# B&R Automation Studio project Tires_Krichev
Automation Studio 3.0.90.25 SP07; Krichev. Equipment tire burning


## Configuration Simulation

### Task classes (Cpu.sw)
```
Cyclic#2:
  spreading <- spreading.prg
  Conv_mitsu <- Conv_mitsubishi.prg [disabled]
  Sleep <- Sleep.prg
  manualCont <- manualControl.prg
  autoContro <- autoControl.prg
  weightCont <- weightControl.prg
  modbusRTU <- modbusRTU.prg
Cyclic#3:
  TechProces <- TechProcess.prg
  visual <- visual.prg
Cyclic#4:
  exampleCpl <- exampleCplusplus.prg [disabled]
DataObjects: Arnc0sys, Acp10sys
NcDataObjects: gmcipsys <- GmcIpConfig.gmcipsys.dob, gmciplbr <- GmcIpConfig.gmciplbr.dob, gmcipcbr <- GmcIpConfig.gmcipcbr.dob, gmciplsm <- GmcIpConfig.gmciplsm.dob, gmcipcsm <- GmcIpConfig.gmcipcsm.dob, gmcipcfg <- GmcIpConfig.gmcipcfg.dob, gmcipiec <- GmcIpConfig.gmcipiec.dob, gmciplog <- GmcIpConfig.gmciplog.dob, gmcipvar <- GmcIpUserConfig.gmcipvar.dob, gmcipfun <- GmcIpUserConfig.gmcipfun.dob, gmcipfub <- GmcIpUserConfig.gmcipfub.dob, gmcipubr <- GmcIpUserConfig.gmcipubr.dob, gmcipusm <- GmcIpUserConfig.gmcipusm.dob
VcDataObjects: Visu <- Visu.dob
Binaries: vccbar, visvc, Visu01, Visu02, vcfntttf, vccshape, vcctext, vccovl, arial, vctcal, vccbtn, vccnum, vcpfar00, vcdsint, vcpdvnc, vcpdsw, vcalarm, vcchspot, vcfile, vcmgr, vccstr, vcresman, vcgclass, vcdsloc, arialbd, vcnet, vcrt, vccalarm, vcclbox, vccbmp, vcbclass, vcshared, vccline, vcctrend, Visu03, Arnc0cfg, Acp10cfg, ashwd, arconfig, sysconf, asfw, iomap
Libraries: AsIecCon, astime, visapi, fileio, dataobj, runtime, standard, dvframe, Arnc0man, AsMem, AsArLog, Acp10man, sys_lib, AsArProf, brsystem, NcGlobal, Acp10par, powerlnk
```

### Acp10cfg.ncc - PLC1/Motion/Acp10cfg.ncc
```
NcConfiguration (Version=2.28.2, NcSwId=acp10)
  ACP10CF1_typ:
    cnt_nettrc_rec_drive = 1500
    bufsize_trace_upload = 1200
    tc_nc_man_task = Cyclic #1
    glob_pv_as_ncobject = Yes
    network_init:
      ncsw_init_execute = Yes
      automatic_execute = No
      node_nr_warning = Yes
      net_err_before_ncact = Yes
    nettrc:
      enter_parsecrec = Yes
      enter_ncaction = Yes
      save_ring_startidx = Yes
```

### Arnc0cfg.ncc - PLC1/Motion/Arnc0cfg.ncc
```
NcConfiguration (Version=1.28.1, NcSwId=arnc0)
  ARNC0CFG_typ:
    sampling_rate = 4000
    cnt_nettrc_rec_drive = 1500
    bufsize_sys_trace = 16#00005000
    enable_mp_log = Yes
    tc_nc_man_task = Cyclic #1
    bg_load = 1
    glob_pv_as_ncobject = Yes
```

## Configuration config

### Task classes (Cpu.sw)
```
Cyclic#4:
  visual <- visual.prg
  TechProces <- TechProcess.prg
  Conv_mitsu <- Conv_mitsubishi.prg [disabled]
  weightCont <- weightControl.prg
  manualCont <- manualControl.prg
  autoContro <- autoControl.prg
  spreading <- spreading.prg
  modbusRTU <- modbusRTU.prg [disabled]
Cyclic#5:
  Sleep <- Sleep.prg
NcDataObjects: gmcipsys <- GmcIpConfig.gmcipsys.dob, gmciplbr <- GmcIpConfig.gmciplbr.dob, gmcipcbr <- GmcIpConfig.gmcipcbr.dob, gmciplsm <- GmcIpConfig.gmciplsm.dob, gmcipcsm <- GmcIpConfig.gmcipcsm.dob, gmcipcfg <- GmcIpConfig.gmcipcfg.dob, gmcipiec <- GmcIpConfig.gmcipiec.dob, gmciplog <- GmcIpConfig.gmciplog.dob, gmcipvar <- GmcIpUserConfig.gmcipvar.dob, gmcipfun <- GmcIpUserConfig.gmcipfun.dob, gmcipfub <- GmcIpUserConfig.gmcipfub.dob, gmcipubr <- GmcIpUserConfig.gmcipubr.dob, gmcipusm <- GmcIpUserConfig.gmcipusm.dob
VcDataObjects: Visu <- Visu.dob
Binaries: vccalarm, vcclbox, vcctext, vcrt, vcchspot, vcpdpp30, vccbar, vcresman, vcpfmtcx, vcptelo, vcfile, vcdsint, vcpdsw, vccshape, arial, vccbmp, vcmgr, Visu01, vcctrend, vcfntttf, vcgclass, vccovl, vctcal, arialbd, vcalarm, vccnum, vccline, vcshared, vcdsloc, vccbtn, vccstr, vcbclass, vcpfpp30, Visu03, Visu02, arconfig, sysconf, ashwd, asfw, iomap
Libraries: fileio, standard, astime, runtime, dataobj, dvframe
```

## Configuration master

### Task classes (Cpu.sw)
```

```

## Configuration slave

### Task classes (Cpu.sw)
same as Physical/master/PLC1/Cpu.sw

- Physical/slave/PLC1/Cpu.per: same as Physical/master/PLC1/Cpu.per
- Physical/slave/PLC1/IoMap.iom: same as Physical/master/PLC1/IoMap.iom
- Physical/slave/PLC1/PvMap.vvm: same as Physical/master/PLC1/PvMap.vvm
## Logical view

### Global.var - Global variables
```iecst
(********************************************************************
 * COPYRIGHT --
 ********************************************************************
 * File: Global.var
 * Author: vzylevich
 * Created: June 24, 2013
 ********************************************************************
 * Global variables of project Tires_Krichev
 ********************************************************************)
VAR
	b : UINT := 0; (*Отладка*)
	a : UINT := 0; (*Отладка*)
	maxTireWeight : USINT := 0; (*Максимальный вес шины*)
	minTireWeight : USINT := 0; (*Минимальный вес шины*)
	pulseSignal : USINT := 0; (*Индикатор запуска пульсирующего сигнала технологического светофора*)
	sensSB4Light : USINT := 0; (*Лампа на кнопке SB4*)
	mod : USINT := 0;
	TON_count : TON := (0);
	TON0 : TON := (0);
	TON_01 : TON := (0);
	count : USINT := 0; (*Счетчик секунд пульсирующего сигнала (30 сек)*)
	var : USINT := 0; (*Переменная для отображения заголовков рольганга*)
	elmotorM : ARRAY[0..12] OF USINT := [13(0)]; (*Массив для электродвигателей*)
	sensRemoteControl : ARRAY[0..13] OF USINT := [14(1)]; (*Массив для датчиков дистанционного управления*)
	sensLocalControl : ARRAY[0..13] OF USINT := [14(0)]; (*Массив для датчиков местного управления (пуск).*)
	sensSQAlarm : ARRAY[0..6] OF USINT := [5(0)]; (*Датчики аварийных предупреждений*)
	sensSQ : ARRAY[0..14] OF USINT := [13(0)]; (*Массив для датчиков положения покрышки на рольгангах и конвейерах.*)
	modeControl : USINT := 0; (*Режим управления*)
	tireWeightRolg7 : USINT := 0; (*Вес шины на рольганге 7*)
	lineCapacityMin : UINT := 0; (*Минимальная производительность линии*)
	lineCapacityMax : UINT := 0; (*Максимальная производительность линии*)
	transporterSpeed : USINT := 0; (*Скорость транспортера*)
	tireWeightMin : USINT := 0; (*Минимальный вес шины, загружаемой на конвейер 8*)
	tireWeightMax : USINT := 0; (*Максимальный вес шины, загружаемой на конвейер 8*)
	furnReady : USINT := 0; (*Готовность печи*)
	tireWeightRolg6 : USINT := 0; (*Вес шины на рольганге 6*)
	tireWeightConv8 : USINT := 0; (*Вес шины на конвейере 8*)
	resValueTires : USINT := 0; (*Остаточное значение шин*)
	realCapacity : USINT := 0; (*Действительное значение производительности*)
	nomCapacity : UINT := 0; (*Номинальное значние производительности*)
	scalesMSG : USINT := 0; (*Сообщение "Весы готовы"*)
	sensSB4 : USINT := 0; (*Датчик автоматического режима управления*)
	sensHL12 : USINT := 0; (*Датчик ручного режима управления*)
	sensY2 : USINT := 0;
	sensY1 : USINT := 0;
END_VAR
(*Датчики*)
VAR
	sensSQ70 : USINT := 0;
	sensSQ68 : USINT := 0;
	sensSQ67 : USINT := 0;
	sensSQ66 : USINT := 0;
	sensSQ65 : USINT := 0;
	sensSQ64 : USINT := 0;
	sensSQ62 : USINT := 0;
	sensSQ51 : USINT := 0;
	sensSQ49 : USINT := 0;
	sensSQ48 : USINT := 0;
	sensSQ46 : USINT := 0;
	sensSQ44 : USINT := 0;
	sensSQ43 : USINT := 0;
	sensSQ42 : USINT := 0;
	sensSQ24 : USINT := 0;
END_VAR
```

- Visualisation Logical/Visu (not shown)

- Visualisation Logical/visual (not shown)

### Program Logical/TechProcess (ANSIC) - the description line work tire burning

#### modesControl.h
```c
/********************************************************************
 * COPYRIGHT --
 ********************************************************************
 * Program: TechProcess
 * File: modesControl.h
 * Author: VZylevich
 * Created: July 05, 2013
 *******************************************************************/

#include <bur/plctypes.h>

#ifdef _DEFAULT_INCLUDES
	#include <AsDefault.h>
#endif

/*Количество датчиков местного управления*/
USINT amountModeControl()
{
	return sizeof(sensRemoteControl);
}

USINT amountSensAlarm()
{
	return sizeof(sensSQAlarm);
}

/*Проверка условий останова автоматического режима*/
BOOL checkAutoStop(USINT array[], USINT numOfElements, BOOL onOff)
{
	for (i = 0; i < numOfElements; i++)
	{
		if (array[i] == onOff)
		{
			checkStop = 0;
			sensSB4 = 0;
			sensSB4Light = 0;
			count = 0;
			TON_count.IN = 0;
			TON_count.ET = 0;
			TON_count.StartTime = 0;
			break;
		}
		else checkStop = 1;
	}
	return checkStop;
}

/*Проверка условий и запуск автоматического режима управления*/
int checkAutoMode()
{
	rControl = checkAutoStop(sensRemoteControl, amountModeControl(), 0);
	sensAlarm = checkAutoStop(sensSQAlarm, amountSensAlarm(), 1);

	if (sensSB4 && rControl && sensAlarm)
	{
		(TON_count.ET < 30000) ? (pulseSignal = 1) : (pulseSignal = 0);	//Пульсирующий сигнал техн. светофоров
		autoMode = 1;
	}
	else
	{
		sensSB4Light = 0;
		count = 0;
		TON_count.IN = 0;
		TON_count.ET = 0;
		TON_count.StartTime = 0;
		autoMode = 0;
	}
	return autoMode;
}

/*Проверка условий и запуск ручного режима управления*/
int checkManMode()
{
	ssModeControl = amountModeControl();
	if (sensHL12 == 1)
	{
		for (i = 0; i < ssModeControl; i++)
			sensLocalControl[i] = 1;
		manMode = 1;
		if (checkAutoMode())
		{
			for (i = 0; i < ssModeControl; i++)
				sensRemoteControl[i] = 0;
			sensSB4 = 0;
			rControl = 0;
			autoMode = 0;
		}
	} else{
		for (i = 0; i < ssModeControl; i++)
			sensLocalControl[i] = 0;
		manMode = 0;
	}
	return manMode;
}

/*int autoMode()
{
	sensSQ[0] ?
	return 0;
}*/
```

#### TechProcess.c - Cyclic code
```c
/********************************************************************
 * COPYRIGHT --
 ********************************************************************
 * Program: TechProcess
 * File: TechProcess.c
 * Author: VZylevich
 * Created: July 02, 2013
 ********************************************************************
 * Implementation of program TechProcess
 ********************************************************************/
#include <bur/plctypes.h>
#include <standard.h>
#include "modesControl.h"

#ifdef _DEFAULT_INCLUDES
	#include <AsDefault.h>
#endif

void _CYCLIC TechProcess(void)
{
	if (checkManMode())
	{
		timeStruct.second = 0;
		foo = 0;
	}
	else if (checkAutoMode())
	{

	}
}
```

#### TechProcess.var - Local variables
```iecst
(********************************************************************
 * COPYRIGHT --
 ********************************************************************
 * Program: TechProcess
 * File: TechProcess.var
 * Author: VZylevich
 * Created: July 02, 2013
 ********************************************************************
 * Local variables of program TechProcess
 ********************************************************************)
VAR
	checkStop : BOOL := FALSE;
	sensAlarm : USINT := 0; (*Датчик предупреждения*)
	rControl : USINT := 0;
	ssModeControl : USINT := 0;
	autoMode : BOOL := FALSE;
	manMode : BOOL := FALSE;
	timeStruct : TIMEStructure := (0);
	foo : UINT := 0; (*Отладка*)
	i : USINT := 0;
END_VAR
```

### Program Logical/Sleep (ANSIC) - A new program

#### Sleep.c - Cyclic code
```c
/********************************************************************
 * COPYRIGHT --
 ********************************************************************
 * Program: Sleep
 * File: Sleep.c
 * Author: VZylevich
 * Created: July 10, 2013
 ********************************************************************
 * Implementation of program Sleep
 ********************************************************************/

#include <bur/plctypes.h>

#ifdef _DEFAULT_INCLUDES
	#include <AsDefault.h>
#endif

_LOCAL USINT i;
_LOCAL USINT foo;

/*Пульсирующий сигнал технологических светофоров длительностью 30 секунд*/
void timerAutoMode(void)
{
	if (sensSB4)
	{
		if(pulseSignal)
		{
			TON_count.IN = !TON_count.Q;
			TON_count.PT = 30000;
			TON(&TON_count);
			if(TON_count.ET < 30000)
			{
				pulseSignal = 1;
				TON_01.IN = !TON_01.Q;
				TON_01.PT = 1000;
				TON(&TON_01);
				count = TON_count.ET / TON_01.PT;
				(count % 2) ? (sensSB4Light = 0) : (sensSB4Light = 1);
			} else
			{
				sensSB4Light = 1;
				pulseSignal = 0;
			}
		}
	}
}

/*Моделирование передвижения шин по конвейеру*/
void tireMoving()
{
	if(foo)
	{
		if(i < sizeof(sensSQ))
		{
			if(i > 0) sensSQ[i-1] = 0;
			sensSQ[i] = 1;
			(i % 2) ? (TON0.IN = 1) : (TON0.IN = 0);
			TON0.PT = 5000;
			TON(&TON0);
			i++;
		}else i = 0;
	}else for(i = 0; i < sizeof(sensSQ); i++)
			sensSQ[i] = 0;
}

void _CYCLIC Sleep(void)
{
	timerAutoMode();
	tireMoving();
}
```

### Program Logical/manualControl (ANSIC) - A new program

#### manualControl.c - Cyclic code
```c
/********************************************************************
 * COPYRIGHT --
 ********************************************************************
 * Program: manualControl
 * File: manualControl.c
 * Author: VZylevich
 * Created: July 15, 2013
 ********************************************************************
 * Implementation of program manualControl
 ********************************************************************/

#include <bur/plctypes.h>

#ifdef _DEFAULT_INCLUDES
	#include <AsDefault.h>
#endif

void _CYCLIC manualControl(void)
{
	/* TODO: Add code here */
}
```

#### modesControl.h
```c
/********************************************************************
 * COPYRIGHT --
 ********************************************************************
 * Program: TechProcess
 * File: modesControl.h
 * Author: VZylevich
 * Created: July 05, 2013
 *******************************************************************/

#include <bur/plctypes.h>

#ifdef _DEFAULT_INCLUDES
	#include <AsDefault.h>
#endif

/*Количество датчиков местного управления*/
USINT amountModeControl()
{
	return sizeof(sensRemoteControl);
}

USINT amountSensAlarm()
{
	return sizeof(sensSQAlarm);
}

/*Проверка условий останова автоматического режима*/
BOOL checkAutoStop(USINT array[], USINT numOfElements, BOOL onOff)
{
	for (i = 0; i < numOfElements; i++)
	{
		if (array[i] == onOff)
		{
			checkStop = 0;
			sensSB4 = 0;
			sensSB4Light = 0;
			count = 0;
			TON_count.IN = 0;
			TON_count.ET = 0;
			TON_count.StartTime = 0;
			break;
		}
		else checkStop = 1;
	}
	return checkStop;
}

/**/
int checkManMode()
{
	ssModeControl = amountModeControl();
	if (sensHL12 == 1)
	{
		for (i = 0; i < ssModeControl; i++)
			sensLocalControl[i] = 1;
		manMode = 1;
		if (checkAutoMode())
		{
			for (i = 0; i < ssModeControl; i++)
				sensRemoteControl[i] = 0;
			sensSB4 = 0;
			rControl = 0;
			autoMode = 0;
		}
	} else{
		for (i = 0; i < ssModeControl; i++)
			sensLocalControl[i] = 0;
		manMode = 0;
	}
	return manMode;
}

/**/
int checkAutoMode()
{
	rControl = checkAutoStop(sensRemoteControl, amountModeControl(), 0);
	sensAlarm = checkAutoStop(sensSQAlarm, amountSensAlarm(), 1);

	if (sensSB4 && rControl && sensAlarm)
	{
		(TON_count.ET < 30000) ? (pulseSignal = 1) : (pulseSignal = 0);
		autoMode = 1;
	}
	else
	{
		sensSB4Light = 0;
		count = 0;
		TON_count.IN = 0;
		TON_count.ET = 0;
		TON_count.StartTime = 0;
		autoMode = 0;
	}
	return autoMode;
}

/*int autoMode()
{
	sensSQ[0] ?
	return 0;
}*/
```

### Program Logical/autoControl (ANSIC) - A new program

#### autoControl.c - Cyclic code
```c
/********************************************************************
 * COPYRIGHT --
 ********************************************************************
 * Program: autoControl
 * File: autoControl.c
 * Author: VZylevich
 * Created: July 15, 2013
 ********************************************************************
 * Implementation of program autoControl
 ********************************************************************/

#include <bur/plctypes.h>

#ifdef _DEFAULT_INCLUDES
	#include <AsDefault.h>
#endif

void _CYCLIC autoControl(void)
{
	/* TODO: Add code here */
}
```

#### modesControl.h
```c
/********************************************************************
 * COPYRIGHT --
 ********************************************************************
 * Program: TechProcess
 * File: modesControl.h
 * Author: VZylevich
 * Created: July 05, 2013
 *******************************************************************/

#include <bur/plctypes.h>

#ifdef _DEFAULT_INCLUDES
	#include <AsDefault.h>
#endif

/*Количество датчиков местного управления*/
USINT amountModeControl()
{
	return sizeof(sensRemoteControl);
}

USINT amountSensAlarm()
{
	return sizeof(sensSQAlarm);
}

/*Проверка условий останова автоматического режима*/
BOOL checkAutoStop(USINT array[], USINT numOfElements, BOOL onOff)
{
	for (i = 0; i < numOfElements; i++)
	{
		if (array[i] == onOff)
		{
			checkStop = 0;
			sensSB4 = 0;
			sensSB4Light = 0;
			count = 0;
			TON_count.IN = 0;
			TON_count.ET = 0;
			TON_count.StartTime = 0;
			break;
		}
		else checkStop = 1;
	}
	return checkStop;
}

/**/
int checkManMode()
{
	ssModeControl = amountModeControl();
	if (sensHL12 == 1)
	{
		for (i = 0; i < ssModeControl; i++)
			sensLocalControl[i] = 1;
		manMode = 1;
		if (checkAutoMode())
		{
			for (i = 0; i < ssModeControl; i++)
				sensRemoteControl[i] = 0;
			sensSB4 = 0;
			rControl = 0;
			autoMode = 0;
		}
	} else{
		for (i = 0; i < ssModeControl; i++)
			sensLocalControl[i] = 0;
		manMode = 0;
	}
	return manMode;
}

/**/
int checkAutoMode()
{
	rControl = checkAutoStop(sensRemoteControl, amountModeControl(), 0);
	sensAlarm = checkAutoStop(sensSQAlarm, amountSensAlarm(), 1);

	if (sensSB4 && rControl && sensAlarm)
	{
		(TON_count.ET < 30000) ? (pulseSignal = 1) : (pulseSignal = 0);
		autoMode = 1;
	}
	else
	{
		sensSB4Light = 0;
		count = 0;
		TON_count.IN = 0;
		TON_count.ET = 0;
		TON_count.StartTime = 0;
		autoMode = 0;
	}
	return autoMode;
}

/*int autoMode()
{
	sensSQ[0] ?
	return 0;
}*/
```

### Program Logical/weightControl (ANSIC) - A new program

#### weightControl.c - Cyclic code
```c
/********************************************************************
 * COPYRIGHT --
 ********************************************************************
 * Program: weightControl
 * File: weightControl.c
 * Author: VZylevich
 * Created: July 15, 2013
 ********************************************************************
 * Implementation of program weightControl
 ********************************************************************/

#include <bur/plctypes.h>

#ifdef _DEFAULT_INCLUDES
	#include <AsDefault.h>
#endif
void _INIT inity(void)
{
	a = 0;
	b = 0;
}

TIME rotationPeriod(void)
{
	/*Определяем время оборота печи*/
	if (sensSQ70){
		rotation = 1;
		time ? (period = time) : (period = 0);
	}
	if (!sensSQ70 && rotation)
		time = clock_ms();

	return period;
}

/*Загрузка печи*/
UDINT furnaceLoading(TIME rotationFurnace)
{
	Qrot = (nomCapacity * (UDINT) rotationFurnace) / hour;
	return Qrot;
}

/*Производительность сжигания*/
UDINT capacityBurning(void)
{
	return (nomCapacity * 1000)/ hour;
}

/*Задержка для успокоения весов*/
void delay(USINT sensor)
{
	if (sensor){
		TON_atten.IN = !TON_atten.Q;
		TON_atten.PT = attenuation;
		TON(&TON_atten);
	}
}
void _CYCLIC weightControl(void)
{
	tRot = rotationPeriod();	//Время одного оборота печи
	if (tRot)
		kgRotation = furnaceLoading(tRot); //Определяем кол-во килограмм шин необходимых для загрузки печи за один оборот
	kgSec = capacityBurning();	//Производительносто подачи шин на сжигание в секунду
	delay(sensSQ70);
	(TON_atten.ET == attenuation) ? (weightMeasure = weight) : (weightMeasure = 0);//Если время успокоения прошло, присвоить значение веса
	if (weightMeasure && !sensSQ[7])	//Если известен вес и на рольганге 7 пусто - включить электродвигатель рольганга
		elmotorM[6] = 1;
	if (weightMeasure && sensSQ[7])		//Если известен вес и на рольганге 7 есть шина, передать измерен. знач. веса шины в загрузку
		loadingRollg7 = weightMeasure;

}
```

#### weightControl.var - Local variables
```iecst
(********************************************************************
 * COPYRIGHT --
 ********************************************************************
 * Program: weightControl
 * File: weightControl.var
 * Author: VZylevich
 * Created: July 15, 2013
 ********************************************************************
 * Local variables of program weightControl
 ********************************************************************)
VAR
	kgSec : USINT := 0; (*Производительность печи*)
	period : USINT := 0;
	rotation : USINT := 0;
	loadingRollg7 : USINT := 0; (*Вес шины на позиции загрузки(рольганг 7)*)
	weight : USINT := 0;
	weightMeasure : USINT := 0;
	TON_atten : TON := (0); (*Время необходимое для успокоения весов перед взвешинванием*)
	attenuation : USINT := 0; (*Затухание весов*)
	Qrot : UDINT := 0;
	kgRotation : REAL := 0.0; (*Кол-во кг сжигаемых шин за 1 оборот*)
END_VAR
VAR CONSTANT
	hour : UDINT := 3600000; (*1 час в мс*)
END_VAR
VAR
	time : TIME := T#0S;
	tRot : TIME := T#0S; (*Время оборота печи*)
	(*TON_weightLoading : TON := (0);*)
END_VAR
```

#### modesControl.h
```c
/********************************************************************
 * COPYRIGHT --
 ********************************************************************
 * Program: TechProcess
 * File: modesControl.h
 * Author: VZylevich
 * Created: July 05, 2013
 *******************************************************************/

#include <bur/plctypes.h>

#ifdef _DEFAULT_INCLUDES
	#include <AsDefault.h>
#endif

/*Количество датчиков местного управления*/
USINT amountModeControl()
{
	return sizeof(sensRemoteControl);
}

USINT amountSensAlarm()
{
	return sizeof(sensSQAlarm);
}

/*Проверка условий останова автоматического режима*/
BOOL checkAutoStop(USINT array[], USINT numOfElements, BOOL onOff)
{
	for (i = 0; i < numOfElements; i++)
	{
		if (array[i] == onOff)
		{
			checkStop = 0;
			sensSB4 = 0;
			sensSB4Light = 0;
			count = 0;
			TON_count.IN = 0;
			TON_count.ET = 0;
			TON_count.StartTime = 0;
			break;
		}
		else checkStop = 1;
	}
	return checkStop;
}

/**/
int checkManMode()
{
	ssModeControl = amountModeControl();
	if (sensHL12 == 1)
	{
		for (i = 0; i < ssModeControl; i++)
			sensLocalControl[i] = 1;
		manMode = 1;
		if (checkAutoMode())
		{
			for (i = 0; i < ssModeControl; i++)
				sensRemoteControl[i] = 0;
			sensSB4 = 0;
			rControl = 0;
			autoMode = 0;
		}
	} else{
		for (i = 0; i < ssModeControl; i++)
			sensLocalControl[i] = 0;
		manMode = 0;
	}
	return manMode;
}

/**/
int checkAutoMode()
{
	rControl = checkAutoStop(sensRemoteControl, amountModeControl(), 0);
	sensAlarm = checkAutoStop(sensSQAlarm, amountSensAlarm(), 1);

	if (sensSB4 && rControl && sensAlarm)
	{
		(TON_count.ET < 30000) ? (pulseSignal = 1) : (pulseSignal = 0);
		autoMode = 1;
	}
	else
	{
		sensSB4Light = 0;
		count = 0;
		TON_count.IN = 0;
		TON_count.ET = 0;
		TON_count.StartTime = 0;
		autoMode = 0;
	}
	return autoMode;
}

/*int autoMode()
{
	sensSQ[0] ?
	return 0;
}*/
```

### Program Logical/dosingTires (ANSIC) - A new program

#### dosingTires.c - Cyclic code
```c
/********************************************************************
 * COPYRIGHT --
 ********************************************************************
 * Program: dosingTires
 * File: dosingTires.c
 * Author: VZylevich
 * Created: July 15, 2013
 ********************************************************************
 * Implementation of program dosingTires
 ********************************************************************/

#include <bur/plctypes.h>

#ifdef _DEFAULT_INCLUDES
	#include <AsDefault.h>
#endif

void _CYCLIC dosingTires(void)
{
	/* TODO: Add code here */
}
```

#### modesControl.h
```c
/********************************************************************
 * COPYRIGHT --
 ********************************************************************
 * Program: TechProcess
 * File: modesControl.h
 * Author: VZylevich
 * Created: July 05, 2013
 *******************************************************************/

#include <bur/plctypes.h>

#ifdef _DEFAULT_INCLUDES
	#include <AsDefault.h>
#endif

/*Количество датчиков местного управления*/
USINT amountModeControl()
{
	return sizeof(sensRemoteControl);
}

USINT amountSensAlarm()
{
	return sizeof(sensSQAlarm);
}

/*Проверка условий останова автоматического режима*/
BOOL checkAutoStop(USINT array[], USINT numOfElements, BOOL onOff)
{
	for (i = 0; i < numOfElements; i++)
	{
		if (array[i] == onOff)
		{
			checkStop = 0;
			sensSB4 = 0;
			sensSB4Light = 0;
			count = 0;
			TON_count.IN = 0;
			TON_count.ET = 0;
			TON_count.StartTime = 0;
			break;
		}
		else checkStop = 1;
	}
	return checkStop;
}

/**/
int checkManMode()
{
	ssModeControl = amountModeControl();
	if (sensHL12 == 1)
	{
		for (i = 0; i < ssModeControl; i++)
			sensLocalControl[i] = 1;
		manMode = 1;
		if (checkAutoMode())
		{
			for (i = 0; i < ssModeControl; i++)
				sensRemoteControl[i] = 0;
			sensSB4 = 0;
			rControl = 0;
			autoMode = 0;
		}
	} else{
		for (i = 0; i < ssModeControl; i++)
			sensLocalControl[i] = 0;
		manMode = 0;
	}
	return manMode;
}

/**/
int checkAutoMode()
{
	rControl = checkAutoStop(sensRemoteControl, amountModeControl(), 0);
	sensAlarm = checkAutoStop(sensSQAlarm, amountSensAlarm(), 1);

	if (sensSB4 && rControl && sensAlarm)
	{
		(TON_count.ET < 30000) ? (pulseSignal = 1) : (pulseSignal = 0);
		autoMode = 1;
	}
	else
	{
		sensSB4Light = 0;
		count = 0;
		TON_count.IN = 0;
		TON_count.ET = 0;
		TON_count.StartTime = 0;
		autoMode = 0;
	}
	return autoMode;
}

/*int autoMode()
{
	sensSQ[0] ?
	return 0;
}*/
```

### Program Logical/bunkerLoad14 (ANSIC) - A new program

#### bunkerLoad14.c - Cyclic code
```c
/********************************************************************
 * COPYRIGHT --
 ********************************************************************
 * Program: bunkerLoad14
 * File: bunkerLoad14.c
 * Author: VZylevich
 * Created: July 15, 2013
 ********************************************************************
 * Implementation of program bunkerLoad14
 ********************************************************************/

#include <bur/plctypes.h>

#ifdef _DEFAULT_INCLUDES
	#include <AsDefault.h>
#endif

void _CYCLIC bunkerLoad14(void)
{
	/* TODO: Add code here */
}
```

#### modesControl.h
```c
/********************************************************************
 * COPYRIGHT --
 ********************************************************************
 * Program: TechProcess
 * File: modesControl.h
 * Author: VZylevich
 * Created: July 05, 2013
 *******************************************************************/

#include <bur/plctypes.h>

#ifdef _DEFAULT_INCLUDES
	#include <AsDefault.h>
#endif

/*Количество датчиков местного управления*/
USINT amountModeControl()
{
	return sizeof(sensRemoteControl);
}

USINT amountSensAlarm()
{
	return sizeof(sensSQAlarm);
}

/*Проверка условий останова автоматического режима*/
BOOL checkAutoStop(USINT array[], USINT numOfElements, BOOL onOff)
{
	for (i = 0; i < numOfElements; i++)
	{
		if (array[i] == onOff)
		{
			checkStop = 0;
			sensSB4 = 0;
			sensSB4Light = 0;
			count = 0;
			TON_count.IN = 0;
			TON_count.ET = 0;
			TON_count.StartTime = 0;
			break;
		}
		else checkStop = 1;
	}
	return checkStop;
}

/**/
int checkManMode()
{
	ssModeControl = amountModeControl();
	if (sensHL12 == 1)
	{
		for (i = 0; i < ssModeControl; i++)
			sensLocalControl[i] = 1;
		manMode = 1;
		if (checkAutoMode())
		{
			for (i = 0; i < ssModeControl; i++)
				sensRemoteControl[i] = 0;
			sensSB4 = 0;
			rControl = 0;
			autoMode = 0;
		}
	} else{
		for (i = 0; i < ssModeControl; i++)
			sensLocalControl[i] = 0;
		manMode = 0;
	}
	return manMode;
}

/**/
int checkAutoMode()
{
	rControl = checkAutoStop(sensRemoteControl, amountModeControl(), 0);
	sensAlarm = checkAutoStop(sensSQAlarm, amountSensAlarm(), 1);

	if (sensSB4 && rControl && sensAlarm)
	{
		(TON_count.ET < 30000) ? (pulseSignal = 1) : (pulseSignal = 0);
		autoMode = 1;
	}
	else
	{
		sensSB4Light = 0;
		count = 0;
		TON_count.IN = 0;
		TON_count.ET = 0;
		TON_count.StartTime = 0;
		autoMode = 0;
	}
	return autoMode;
}

/*int autoMode()
{
	sensSQ[0] ?
	return 0;
}*/
```

### Program Logical/furnaceLoading (ANSIC) - A new program

#### furnaceLoading.c - Cyclic code
```c
/********************************************************************
 * COPYRIGHT --
 ********************************************************************
 * Program: furnaceLoading
 * File: furnaceLoading.c
 * Author: VZylevich
 * Created: August 01, 2013
 ********************************************************************
 * Implementation of program furnaceLoading
 ********************************************************************/

#include <bur/plctypes.h>

#ifdef _DEFAULT_INCLUDES
	#include <AsDefault.h>
#endif

void _CYCLIC furnaceLoading(void)
{
	/* TODO: Add code here */
}
```

### Program Logical/spreading (ANSIC) - A new program

#### spreading.c - Cyclic code
```c
/********************************************************************
 * COPYRIGHT --
 ********************************************************************
 * Program: spreading
 * File: spreading.c
 * Author: VZylevich
 * Created: July 16, 2013
 ********************************************************************
 * Implementation of program spreading
 ********************************************************************/

#include <bur/plctypes.h>

#ifdef _DEFAULT_INCLUDES
	#include <AsDefault.h>
#endif

void _INIT init()
{
	n = 1;
	spreadingStart = 0;
	spreadingStop = 0;
}
/*Задержка времени для растягивания шины */
TIME spreadingDelay()
{
	TON_spreading.IN = !TON_spreading.Q;
	TON_spreading.PT = tp;
	TON(&TON_spreading);
	return TON_spreading.ET;
}

/*Проверка загрузки рольганга*/
INT checkLoadTires(int i, int k)
{
	if(sensSQ[i] & !sensSQ[k])
		rolgMoving[k-1] = 1;
	return rolgMoving[k-1];
}
/*Участок растаскивания шин*/
void spreadingPlot(int prev, int current)
{
	if(!sensSQ[current] && checkLoadTires(prev, current))
	{
		elmotorM[current-1] = 1;
		TON_spreading_repeat.IN = !TON_spreading_repeat.Q;
		TON_spreading_repeat.PT = tp2;
		TON(&TON_spreading_repeat);
		if(TON_spreading_repeat.ET >= tp2)
		{
			spreadingStart = 1;
			spreadingStop = 0;
			TON_spreading.ET = 0;
		}
		if(!spreadingStop)
		{
			elmotorM[prev-1] = 1;
			spreadingStart = 1;
		} else spreadingStart = 0;
	} else
	{
		elmotorM[current-1] = 0;
		rolgMoving[current-1] = 0;
		spreadingStart = 0;
	}
	if(spreadingStart && (TON_spreading.ET < tp))
	{
		TON_spreading.IN = !TON_spreading.Q;
		TON_spreading.PT = tp;
		TON(&TON_spreading);
	}else
	{
		elmotorM[prev-1] = 0;
		spreadingStop = 1;
	}
}

void _CYCLIC spreading(void)
{
	/*Включить рольганг, если шины загружены и растаскивать, пока не включится SQ22*/
	if(!sensSQ[1] & checkLoadTires(0, 1))
		elmotorM[0] = 1;
	else
	{
		elmotorM[0] = 0;
		rolgMoving[0] = 0;
	}

	rolgangCycle = sizeof(rolgMoving);
	if((n >= rolgangCycle) )
		n = 1;
	if(n < rolgangCycle)
	{
		spreadingPlot(n, n+1);
		if(sensSQ[n+1])
		{
			n++;
			spreadingStop = 0;
			TON_spreading.ET = 0;
		}
	}
}
```

#### spreading.var - Local variables
```iecst
(********************************************************************
 * COPYRIGHT --
 ********************************************************************
 * Program: spreading
 * File: spreading.var
 * Author: VZylevich
 * Created: July 16, 2013
 ********************************************************************
 * Local variables of program spreading
 ********************************************************************)
VAR
	rolgangCycle : USINT := 0;
	n : USINT := 1; (*spreadingPlotDone : USINT := 0; (*Участок растаскивания*) (*elapsedTime : TIME := T#0S;*)
	tp2 : TIME := 2; (*Время движения шины по конвейеру*)
	tp : TIME := T#03S; (*Время, в течение которого шина надвигается частично на следующий рольганг*)
END_VAR
(*startRolg : USINT := 0; (*Контроль поступления шин на рольганг 1 - сигнал датчика SQ1-SQ22, включение рольганга*)
VAR
	TON_spreading_repeat : TON := (0);
	TON_spreading : TON := (0);
	spreadingStop : USINT;
	spreadingStart : USINT := 0;
	rolgMoving : ARRAY[0..6] OF USINT := [7(0)];
END_VAR
```

### Program Logical/Conv_mitsubishi (ANSIC) - rs_485

#### hp.h
```c
typedef
struct sHP
{
  struct sHP_in /* входные данные*/
  {
  	/* частотники */

	REAL Con1_Fr;	/* Задание частоты для преобразователя №1 */
	REAL Con1_F;  	/* Выходная частота преобразователя №1 */
	REAL Con1_U;  	/* Выходное напряжение преобразователя №1 */
	REAL Con1_I;  	/* Выходной ток преобразователя №1 */

    REAL Con2_Fr; 	/* Задание частоты для преобразователя №2 */
	REAL Con2_F;  	/* Выходная частота преобразователя №2 */
	REAL Con2_U;  	/* Выходное напряжение преобразователя №2 */
	REAL Con2_I;  	/* Выходной ток преобразователя №2 */

	REAL Con3_Fr; 	/* Задание частоты для преобразователя №3 */
	REAL Con3_F;  	/* Выходная частота преобразователя №3 */
	REAL Con3_U;  	/* Выходное напряжение преобразователя №3 */
	REAL Con3_I;  	/* Выходной ток преобразователя №3 */

	REAL Con4_Fr; 	/* Задание частоты для преобразователя №4 */
	REAL Con4_F;  	/* Выходная частота преобразователя №4 */
	REAL Con4_U;  	/* Выходное напряжение преобразователя №4 */
	REAL Con4_I;  	/* Выходной ток преобразователя №4 */

		REAL Con5_Fr; 	/* Задание частоты для преобразователя №5 */
		REAL Con5_F;  	/* Выходная частота преобразователя №5 */
		REAL Con5_U;  	/* Выходное напряжение преобразователя №5 */
		REAL Con5_I;  	/* Выходной ток преобразователя №5 */

		REAL Con6_Fr; 	/* Задание частоты для преобразователя №6 */
		REAL Con6_F;  	/* Выходная частота преобразователя №6 */
		REAL Con6_U;  	/* Выходное напряжение преобразователя №6 */
		REAL Con6_I;  	/* Выходной ток преобразователя №6 */

  } in;

  struct sHP_out /* выходные данные*/
  {
		REAL Con1_Fr;	/* Задание частоты для преобразователя №1 */
	    REAL Con2_Fr; 	/* Задание частоты для преобразователя №2 */
		REAL Con3_Fr; 	/* Задание частоты для преобразователя №3 */
		REAL Con4_Fr; 	/* Задание частоты для преобразователя №4 */
		REAL Con5_Fr; 	/* Задание частоты для преобразователя №5 */
		REAL Con6_Fr; 	/* Задание частоты для преобразователя №6 */

  } out;
} HP_data;

/*--------------------------------------------------------------------*/
```

#### omron.c
```c
#include <bur/plc.h>
#include <bur/plctypes.h>
#include <string.h>
#include "hp.h"
#include <dvframe.h>

/*********************** Объявление GLOBAL и LOCAL переменных *****************************/

/*_GLOBAL HP_data RunHP;	 структура для контроллера
_LOCAL HP_data UsrHP;	 структура для панели

_GLOBAL FRM_xopen_typ FrameXOpenStruct;
_GLOBAL XOPENCONFIG   XOpenConfigStruct;
_GLOBAL FRM_gbuf_typ  FrameGetBufferStruct;
_GLOBAL FRM_rbuf_typ  FrameReleaseBufferStruct;
_GLOBAL FRM_robuf_typ FrameReleaseOutputBufferStruct;
_GLOBAL FRM_write_typ FrameWriteStruct;
_GLOBAL FRM_read_typ  FrameReadStruct;
_GLOBAL UINT   		 StatusOpen, StatusWrite, StatusRead, StatusGetBuffer, StatusReleaseBuffer;
_GLOBAL UINT   		 SendBufferLength, ReadBufferLength, StatusReleaseOutputBuffer;
_GLOBAL UDINT  		 Ident;
_GLOBAL UDINT* 		 SendBuffer;
_GLOBAL UDINT* 		 ReadBuffer;
_GLOBAL USINT  		 T[8], T1[8],R[13], Error, leng, step;
_GLOBAL BOOL 		    status_read;
_GLOBAL REAL 		    F[5], Fr[5], U[5], I[5];
//_GLOBAL STRING   		 StringDevice[30], StringMode[30]; */

_GLOBAL   REAL 		    F[6], Fr[6], U[6], I[6],Con_Fr[6];
_LOCAL   BOOL 		    status_read;
_LOCAL  UDINT  		 Ident;
_LOCAL  UDINT* 		 SendBuffer;
_LOCAL  UDINT* 		 ReadBuffer;
_LOCAL  FRM_xopen_typ FrameXOpenStruct;
_LOCAL XOPENCONFIG   XOpenConfigStruct;
_LOCAL  FRM_gbuf_typ  FrameGetBufferStruct;
_LOCAL FRM_rbuf_typ  FrameReleaseBufferStruct;
_LOCAL  FRM_robuf_typ FrameReleaseOutputBufferStruct;
_LOCAL  FRM_write_typ FrameWriteStruct;
_LOCAL  FRM_read_typ  FrameReadStruct;
_LOCAL UINT   		 StatusOpen, StatusWrite, StatusRead, StatusGetBuffer, StatusReleaseBuffer;
_LOCAL UINT   		 SendBufferLength, ReadBufferLength, StatusReleaseOutputBuffer;
_LOCAL USINT  		 T[8], T1[8],R[13], Error, leng, step;
_GLOBAL   HP_data   RunHP;
_LOCAL    HP_data   UsrHP;
_LOCAL STRING  		 StringDevice[30], StringMode[30];
//_GLOBAL  UINT transporterSpeed;
void _INIT Init()
{
	memset(&T, 0, sizeof(T));
	memset(&R, 0, sizeof(R));
	memset(&F, 0, sizeof(F));
	memset(&Fr, 0, sizeof(Fr));
	memset(&U, 0, sizeof(U));
	memset(&I, 0, sizeof(I));
	memset(&T1, 0, sizeof(T1));
	status_read = 0;
	step = 1;
	leng = sizeof(T);
	Error = 0;
	strcpy(StringDevice, "SS1.IF2");
	strcpy(StringMode, "PHY=RS485 /BD=9600 /PA=E /DB=8 /SB=1");

	XOpenConfigStruct.idle     = 4;
	XOpenConfigStruct.delimc   = 0;
	XOpenConfigStruct.delim[0] = 0;
	XOpenConfigStruct.delim[1] = 0;
	XOpenConfigStruct.tx_cnt   = 2;
	XOpenConfigStruct.rx_cnt   = 2;
	XOpenConfigStruct.tx_len   = 256;
	XOpenConfigStruct.rx_len   = 256;
	XOpenConfigStruct.argc     = 0;
	XOpenConfigStruct.argv     = 0;

	FrameXOpenStruct.device = (UDINT) StringDevice;
	FrameXOpenStruct.mode   = (UDINT) StringMode;
	FrameXOpenStruct.config = (UDINT) &XOpenConfigStruct;
	FrameXOpenStruct.enable = 1;

	FRM_xopen(&FrameXOpenStruct);
	StatusOpen = FrameXOpenStruct.status;
	Ident = FrameXOpenStruct.ident;

	if (StatusOpen != 0)
	{
		Error = 1;
	}
}

UINT CRC(USINT *data, int length)
{
	int i, j;
	UINT CRC = 0xFFFF, bit;

	for (i = 0; i < length; i++)
	{
		CRC ^= (UINT)data[i];

		for (j = 0; j < 8 ; j++)
		{
			bit = CRC & 0x0001;
			CRC >>= 1;
			if (bit) CRC ^= 0xA001;
		}
	}
	return CRC;
}
/*функция записи команды для ПЧ при записи и чтении по Modbus RTU */
void Write(USINT s,USINT Icode,USINT A1,USINT A2,USINT D1,USINT D2)
{
	FrameGetBufferStruct.enable = 1;
	FrameGetBufferStruct.ident  = Ident;
	FRM_gbuf(&FrameGetBufferStruct);
	SendBuffer = (UDINT*) FrameGetBufferStruct.buffer;
	SendBufferLength = FrameGetBufferStruct.buflng;
	StatusGetBuffer  = FrameGetBufferStruct.status;

	if (StatusGetBuffer == 0)
	{
		T[0]  = s;	    /*номер инвертора*/
		T[1]  = Icode;  /* код инструкции 0x03 или 0х06*/
		T[2]  = A1;	 /*начальный адрес Н/адрес регистра H*/
		T[3]  = A2;	 /*начальный адрес L/адрес регистра L*/
		T[4]  = D1;	 /*количество адресов Н/данные Н*/
		T[5]  = D2;	 /* количество адресов L/данные L*/
		T[6]  = 0x00;	 /*контрольная сумма L*/
		T[7]  = 0x00;	 /* контрольная сумма H*/

		*(UINT *)(T + sizeof(T) - 2) = CRC(T, sizeof(T) - 2);
		memcpy(SendBuffer, T, sizeof (T));

		status_read = 1;

		FrameWriteStruct.ident  = Ident;
		FrameWriteStruct.buffer = (UDINT) SendBuffer;
		FrameWriteStruct.buflng = sizeof (T);
		FrameWriteStruct.enable = 1;
		FRM_write(&FrameWriteStruct);
		StatusWrite = FrameWriteStruct.status;

		if (StatusWrite != 0)
		{
			FrameReleaseOutputBufferStruct.enable = 1;
			FrameReleaseOutputBufferStruct.ident  = Ident;
			FrameReleaseOutputBufferStruct.buffer = (UDINT) SendBuffer;
			FrameReleaseOutputBufferStruct.buflng = SendBufferLength;
			FRM_robuf(&FrameReleaseOutputBufferStruct);
			StatusReleaseOutputBuffer = FrameReleaseOutputBufferStruct.status;
			Error = 3;

			if (StatusReleaseOutputBuffer != 0)
			{
				Error = 4;
			}
		}
	}
	else
	{
		Error = 2;
	}
}
/*функция чтения ПЧ при чтении частоты,тока и напряжения (03)*/
void Read()
{
	USINT rr = 0;
	USINT B[2];
	FrameReadStruct.enable = 1;
	FrameReadStruct.ident = Ident;

	FRM_read(&FrameReadStruct);

	ReadBuffer = (UDINT*) FrameReadStruct.buffer;
	ReadBufferLength = FrameReadStruct.buflng;
	StatusRead = FrameReadStruct.status;

	if (StatusRead == 0)
	{
		memset(&B, 0, sizeof(B));
		memcpy(R, ReadBuffer, sizeof(R));
		*(UINT *)B = CRC(R, sizeof(R) - 2);
		if ((B[0] == R[11])&&(B[1] == R[12]))
		{
			rr = R[0];
			F[rr]  = 256*R[3] + R[4];
			I[rr]  = 256*R[5] + R[6];
			U[rr]  = 256*R[7] + R[8];

		}
		FrameReleaseBufferStruct.enable = 1;
		FrameReleaseBufferStruct.ident  = Ident;
		FrameReleaseBufferStruct.buffer = (UDINT) ReadBuffer;
		FrameReleaseBufferStruct.buflng = ReadBufferLength;
		FRM_rbuf(&FrameReleaseBufferStruct);
		StatusReleaseBuffer = FrameReleaseBufferStruct.status;

		if (StatusReleaseBuffer != 0)
		{
			Error = 5;
		}
	}
	else
	{
		Error = 6;
	}

}
/*функция чтения ПЧ при записи заданной частоты (06)*/
void Read_W()
{
	USINT rr = 0;
	USINT B[2];
	FrameReadStruct.enable = 1;
	FrameReadStruct.ident = Ident;

	FRM_read(&FrameReadStruct);

	ReadBuffer = (UDINT*) FrameReadStruct.buffer;
	ReadBufferLength = FrameReadStruct.buflng;
	StatusRead = FrameReadStruct.status;

	if (StatusRead == 0)
	{
		memset(&B, 0, sizeof(B));
		memcpy(R, ReadBuffer, sizeof(R));
		*(UINT *)B = CRC(R, sizeof(R) - 2);
		if ((B[0] == R[11])&&(B[1] == R[12]))
		{

			rr = R[0];
			Fr[rr] = 256*R[4] + R[5];
		}
		FrameReleaseBufferStruct.enable = 1;
		FrameReleaseBufferStruct.ident  = Ident;
		FrameReleaseBufferStruct.buffer = (UDINT) ReadBuffer;
		FrameReleaseBufferStruct.buflng = ReadBufferLength;
		FRM_rbuf(&FrameReleaseBufferStruct);
		StatusReleaseBuffer = FrameReleaseBufferStruct.status;

		if (StatusReleaseBuffer != 0)
		{
			Error = 5;
		}
	}
	else
	{
		Error = 6;
	}
}
/*функция чтения ПЧ по Modbus RTU */
void Read_R()
{
	if (step <= 6)
	{
		if (!status_read)
		{	T1[1]=0x03;
			T1[2]=0x00;
			T1[3]=0xc8;
			T1[4]=0x00;
			T1[5]=0x04;
			Write(step, T1[1] , T1[2],T1[3],T1[4],T1[5]);
		}
		else
		{
			Read();
			status_read = 0;

			RunHP.in.Con1_F = F[1]*0.01;
			RunHP.in.Con1_U = U[1]*0.1;
			RunHP.in.Con1_I = I[1]*0.1;

			RunHP.in.Con2_F = F[2]*0.01;
			RunHP.in.Con2_U = U[2]*0.1;
			RunHP.in.Con2_I = I[2]*0.1;

			RunHP.in.Con3_F = F[3]*0.01;
			RunHP.in.Con3_U = U[3]*0.1;
			RunHP.in.Con3_I = I[3]*0.1;

			RunHP.in.Con4_F = F[4]*0.01;
			RunHP.in.Con4_U = U[4]*0.1;
			RunHP.in.Con4_I = I[4]*0.1;

			RunHP.in.Con5_F = F[5]*0.01;
			RunHP.in.Con5_U = U[5]*0.1;
			RunHP.in.Con5_I = I[5]*0.1;

			RunHP.in.Con6_F = F[6]*0.01;
			RunHP.in.Con6_U = U[6]*0.1;
			RunHP.in.Con6_I = I[6]*0.1;
			step++;
		}
	}
	else step = 1;

}
	/*функция записи Fr в ПЧ по Modbus RTU */
void Write_Fr()
{   Con_Fr[1]=RunHP.out.Con1_Fr;
	Con_Fr[2]=RunHP.out.Con2_Fr;
	Con_Fr[3]=RunHP.out.Con3_Fr;
	Con_Fr[4]=RunHP.out.Con4_Fr;
	Con_Fr[5]=RunHP.out.Con5_Fr;
	Con_Fr[6]=RunHP.out.Con6_Fr;
	if (step <= 6)
	{
		if (!status_read)
		{	T1[1]=0x06;
			T1[2]=0x00;
			T1[3]=0x0d;
			T1[4]=Con_Fr[step]*100 / 256;
			T1[5]=Con_Fr[step]*100-T1[4]*256;

			Write(step, T1[1] , T1[2],T1[3],T1[4],T1[5]);
		}
		else
		{
			Read_W();
			status_read = 0;
			RunHP.in.Con1_Fr = Fr[1]*0.01;
			RunHP.in.Con2_Fr = Fr[2]*0.01;
			RunHP.in.Con3_Fr = Fr[3]*0.01;
			RunHP.in.Con4_Fr = Fr[4]*0.01;
			RunHP.in.Con5_Fr = Fr[5]*0.01;
			RunHP.in.Con6_Fr = Fr[6]*0.01;
			step++;
		}
	}
	else step = 1;

}

void _CYCLIC run()
{
	UsrHP.in=RunHP.in;
	//RunHP.out.Con1_Fr=transporterSpeed;
	Write_Fr();
	Read_R();
}
```

### Program Logical/modbusRTU (ANSIC)

#### modbusRTU.var
```iecst
VAR
	B1 : ARRAY[0..1] OF USINT := [2(0)];
	e : USINT := 0;
	state : USINT := 0; (*0 - нет действий, 1 - запись, 2 - чтение, 3 - чтение + верное CRC*)
	alarm : USINT := 0; (*0 - нет аварий, 1 - не записал, 2 - не считал, 3 - не успешно записал, 4 - не совпало CRC при чтении*)
END_VAR
```

#### modbusRTU.c
```c
#include <bur/plc.h>
#include <bur/plctypes.h>

#include <string.h>
#include <dvframe.h>

#ifdef _DEFAULT_INCLUDES
 #include <AsDefault.h>
#endif

/* Энергосоюз ЦП9010 */
_LOCAL FRM_xopen_typ 	mbXOpenStruct;
_LOCAL XOPENCONFIG   	XOpenConfigStruct;
_LOCAL FRM_gbuf_typ  	mbGetBufferStruct;
_LOCAL FRM_rbuf_typ  	mbReleaseBufferStruct;
_LOCAL FRM_robuf_typ 	mbReleaseOutputBufferStruct;
_LOCAL FRM_write_typ 	mbWriteStruct;
_LOCAL FRM_read_typ  	mbReadStruct;

_LOCAL STRING StringDevice[30], StringMode[40];

_LOCAL USINT Tb[8], Rb[61];
_LOCAL BOOL enable;

void _INIT modbusRTUINIT( void ){
	memset(&Tb, 0, sizeof(Tb));
	memset(&Rb, 0, sizeof(Rb));
	enable = 1;

	strcpy(StringDevice, "SS1.IF2");
  	strcpy(StringMode, "PHY=RS485 /BD=9600 /PA=N /DB=8 /SB=1");

	XOpenConfigStruct.idle     = 4;
	XOpenConfigStruct.delimc   = 0;
	XOpenConfigStruct.delim[0] = 0;
	XOpenConfigStruct.delim[1] = 0;
	XOpenConfigStruct.tx_cnt   = 2;
	XOpenConfigStruct.rx_cnt   = 2;
	XOpenConfigStruct.tx_len   = 256;
	XOpenConfigStruct.rx_len   = 256;
	XOpenConfigStruct.argc     = 0;
	XOpenConfigStruct.argv     = 0;

	mbXOpenStruct.device = (UDINT) StringDevice;
	mbXOpenStruct.mode   = (UDINT) StringMode;
	mbXOpenStruct.config = (UDINT) &XOpenConfigStruct;
	mbXOpenStruct.enable = 1;

	FRM_xopen(&mbXOpenStruct);
	//Передать вес нетто - c2h; обнулить показания веса - c0h
	Tb[0]  	= 0xff;
   	Tb[1]  	= 0xC2;
    Tb[2]  	= 0x01;
    Tb[3]	= 0x03;
	Tb[4]	= 0x00;
    Tb[5]	= 0x1c;
    Tb[6]	= 0x00;
    Tb[7]	= 0x00;
}

/* Подсчет CRC, ModBus RTU */
UINT CRC(USINT *data, USINT length){
	int i, j;
  	UINT CRC = 0xFFFF, bit;

	for (i = 0; i < length; i++){
    	CRC ^= (UINT)data[i];
    	for (j = 0; j < 8 ; j++){
      		bit = CRC & 0x0001;
      		CRC >>= 1;
      		if (bit) CRC ^= 0xA001;
    	}
	}
	return CRC;
}

/* Функция Write, запись в буфер */
void Write(){
	mbGetBufferStruct.enable = 1;
    mbGetBufferStruct.ident  = mbXOpenStruct.ident;
    FRM_gbuf(&mbGetBufferStruct);

	if (!mbGetBufferStruct.status){
//		Tb[0]  	= 0xff;
//    	Tb[1]  	= 0x04;
//      Tb[2]  	= 0x01;
//      Tb[3]	= 0x03;
//      Tb[4]	= 0x00;
//      Tb[5]	= 0x1c;
		Tb[6]	= 0x00;
      	Tb[7]	= 0x00;
		*(UINT *)(Tb + sizeof(Tb) - 2) = CRC(Tb, sizeof(Tb) - 2);
        *(UINT *)B1 = CRC(Tb, sizeof(Tb) - 2);

		memcpy( (USINT*) mbGetBufferStruct.buffer, Tb, sizeof (Tb));
		state	= 1;
		mbWriteStruct.ident  = mbXOpenStruct.ident;
        mbWriteStruct.buffer = (UDINT) mbGetBufferStruct.buffer;
        mbWriteStruct.buflng = sizeof(Tb);
        mbWriteStruct.enable = 1;
        FRM_write(&mbWriteStruct);

        if (mbWriteStruct.status != 0){
       		alarm = 3;
        	mbReleaseOutputBufferStruct.enable = 1;
            mbReleaseOutputBufferStruct.ident  = mbXOpenStruct.ident;
            mbReleaseOutputBufferStruct.buffer = (UDINT) mbGetBufferStruct.buffer;
            mbReleaseOutputBufferStruct.buflng = mbGetBufferStruct.buflng;
            FRM_robuf(&mbReleaseOutputBufferStruct);
        }
    } else alarm = 1;
}

/* Функция Read, чтение из буфера */
void Read(){
	USINT B[2];
 	mbReadStruct.enable = 1;
    mbReadStruct.ident 	= mbXOpenStruct.ident;
    FRM_read(&mbReadStruct);
	memset(&Rb, 0, sizeof(Rb) );

    if (!mbReadStruct.status){
   		memset(&B, 0, sizeof(B));
		memcpy(Rb, (USINT*) mbReadStruct.buffer, sizeof(Rb) );
        *(UINT *)B = CRC(Rb, sizeof(Rb) - 2);
		state	= 2;
		/* Проверка CRC */
		if( (B[0] == Rb[59]) && (B[1] == Rb[60])){
       	    state	= 3;
       	    e 		= 0;

			/* формирование аналоговых параметров */
			rs485[0].D 	= Rb[3]*256 + Rb[4];
			rs485[1].D 	= Rb[5]*256 + Rb[6];
			rs485[2].D 	= Rb[7]*256 + Rb[8];
			rs485[3].D 	= Rb[9]*256 + Rb[10];
			rs485[4].D 	= Rb[11]*256 + Rb[12];
			rs485[5].D 	= Rb[13]*256 + Rb[14];
			rs485[6].D 	= Rb[15]*256 + Rb[16];
			rs485[7].D 	= Rb[17]*256 + Rb[18];
			rs485f		= (Rb[19]*256 + Rb[20]) * 50 / 50000;
			rs485cos	= (Rb[21]*256 + Rb[22]) / 1000;
			rs485[8].D = Rb[23]*256 + Rb[24];
			rs485[9].D = Rb[25]*256 + Rb[26];
			rs485[10].D = Rb[27]*256 + Rb[28];
			rs485[11].D = Rb[29]*256 + Rb[30];
			rs485[12].D = Rb[31]*256 + Rb[32];
			rs485[13].D = Rb[33]*256 + Rb[34];
			rs485[14].D = Rb[35]*256 + Rb[36];
			rs485[15].D = Rb[37]*256 + Rb[38];
			rs485[16].D = Rb[39]*256 + Rb[40];
			rs485[17].D = Rb[41]*256 + Rb[42];
			rs485[18].D = Rb[43]*256 + Rb[44];
			rs485[19].D = Rb[45]*256 + Rb[46];
			rs485[20].D = Rb[47]*256 + Rb[48];
			rs485[21].D = Rb[49]*256 + Rb[50];
			rs485[22].D = Rb[51]*256 + Rb[52];
			rs485cosa	= (Rb[53]*256 + Rb[54]) / 1000;
			rs485cosb	= (Rb[55]*256 + Rb[56]) / 1000;
			rs485cosc	= (Rb[57]*256 + Rb[58]) / 1000;
		} else{
			e++;
			if(2 < e){
				alarm = 4;
				e = 3;
			}
		}

     	mbReleaseBufferStruct.enable = 1;
     	mbReleaseBufferStruct.ident  = mbXOpenStruct.ident;
     	mbReleaseBufferStruct.buffer = mbReadStruct.buffer;
     	mbReleaseBufferStruct.buflng = mbReadStruct.buflng;
     	FRM_rbuf(&mbReleaseBufferStruct);
     } else alarm = 2;
}

/* Функция реализации процесса обмена по ModBus */
void mb_main(void){
	if (enable){
		state = 0;
		alarm = 0;
		Write();
		if (state == 1) Read();

		/* отработка аварии !alarm */
		if ((alarm > 0) && !sim){
			memset(&Rb, 0, sizeof(Rb) );
			memset(&rs485, 0, sizeof(rs485));
			rs485f = 0;
			rs485cos = rs485cosa = rs485cosb = rs485cosc = 0;
			rs485f_St	= 6;
			rs485cos_St	= 6;
			rs485_alarm = 1;
		}
		else {
			if (rs485f < 49) rs485f_St = 3;
			else if (rs485f > 51) rs485f_St = 4;
			else rs485f_St = 0;
			rs485cos_St	= 0;
			rs485_alarm	= 0;

		}
	} else{
  		state = 0;
  		alarm = 0;
	}
}

void _CYCLIC modbusRTUCYCLIC( void ){
	mb_main();
}
```

#### dac.typ - Local data types
```iecst
TYPE
	aiS_typ : 	STRUCT  (*Структура характеристик AI, i/o*)
		D : INT; (*PV*)
	END_STRUCT;
END_TYPE
```

#### cp10.var - Local variables
```iecst
(*Структуры параметров аналоговых входных величин для уставки*)
VAR
	sim : BOOL := FALSE;
	rs485_alarm : BOOL := FALSE;
	rs485 : ARRAY[0..22] OF aiS_typ := [23(0)];
	rs485f : REAL := 0.0;
	rs485f_St : USINT := 0;
	rs485cos : INT := 0;
	rs485cosa : INT := 0;
	rs485cosb : INT := 0;
	rs485cosc : INT := 0;
	rs485cos_St : USINT := 0;
END_VAR
```

### Program Logical/exampleCplusplus (ANSIC) - A new program

#### exampleCplusplus.c - Cyclic code
```c
/********************************************************************
 * COPYRIGHT --
 ********************************************************************
 * Program: exampleCplusplus
 * File: exampleCplusplus.c
 * Author: VZylevich
 * Created: August 12, 2013
 ********************************************************************
 * Implementation of program exampleCplusplus
 ********************************************************************/

#include <bur/plctypes.h>
//#include <stdafx.h>
#include <stdio.h>
#include <iostream>
#include <string.h>
//#include <conio.h>

#ifdef _DEFAULT_INCLUDES
	#include <AsDefault.h>
#endif

unsigned char CRCMaker(unsigned char b_input, unsigned char b_CRC)
{
	_asm
	{
		mov al,b_input
		mov ah,b_CRC
		mov cx,8
		mod1:  rol al,1
		rcl ah,1
		jnc mod2
		xor ah,69h
			mod2:  dec cx
		jnz mod1
		mov b_CRC,ah
	}
	return b_CRC;
}

void _CYCLIC exampleCplusplus(void)
{
	//using namespace std;
	unsigned char crc=0x00;
	unsigned char request[3]={0x01, 0xC2, 0x00}; //Запрос передать вес нетто, команда 0xC2

	for (int i=0; i<=2; i++)
		{
		crc=CRCMaker(request[i],crc); //расчёт контрольной суммы для посылаемого запроса
	}
	//Добавив разделители (байт FF в начале и 2 байта FF в конце сообщения), получаем запрос - байтовый массив длинной 5 байт, массив нужно передать ТВ003/05H
	cout<< "Request to TB3: "<<std::hex<<255<<" "<<int(request[0])<<" "<<int(request[1])<<" "<<int(crc)<<" "<<255<<" "<<255<<endl;

		//Наример ТВ003/05H ответил так FF 01 C2 40 14 00 B0 D2 FF FF
		//Проверим принятое ли сообщение без ошибок
		unsigned char answer[7]={0x01, 0xC2, 0x40, 0x14, 0x00, 0xB0, 0xD2};
	crc=0x00;
	cout<< "Answer from TB3: "<<std::hex<<255<<" ";
	for (int i=0; i<=6; i++)
		{
		cout<<int(answer[i])<<" ";
			crc=CRCMaker(answer[i],crc); //проверка контрольной суммы сообщения, полученного от ТВ003/05H
	}
	cout<<255<<" "<<255<<endl;

	if (int(crc)==0)
	{
		cout<< "Answer from TB3 received successfully!"<<endl; //принято без ошибок
	}
	else
	{
		cout<< "Answer from TB3 received with errors!"<<endl; //принято с ошибками
		};

	getch();
	return 0;
}
```

Listed in the project but not available here: Logical/Libraries, Logical/GmcIpConfig, Logical/GmcIpUserConfig
